FUNCTION_BLOCK REGRESS_OUT (* HMI elements for outputs of a REGRESS instance *)
  (* Standard: IEC 61499; Classification: HMI; Function: Output; Type: Linear Regression *)
  (* Version 0.0, 2006-07-20, JHC, Holobloc Inc *)
  (* Compiler header: package fb.rt.hmi; *)
  (* Compiler Java Sun JDK 1.5.0 *)
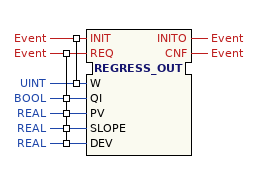
  EVENT_INPUT
    INIT WITH W; (* Initialization Request *)
    REQ WITH QI, PV, SLOPE, DEV; (* Request to Display Data *)
  END_EVENT
  EVENT_OUTPUT
    INITO; (* Initialization Confirm *)
    CNF; (* Data Display Confirmation *)
  END_EVENT
  VAR_INPUT
    W : UINT := 10; (* Text field width in characters *)
    QI : BOOL; (* Sample buffer full, outputs valid *)
    PV : REAL; (* Projected next value of regressed data *)
    SLOPE : REAL; (* Slope of regressed data, IN units per clock period. *)
    DEV : REAL; (* Estimated standard deviation from regression line *)
  END_VAR
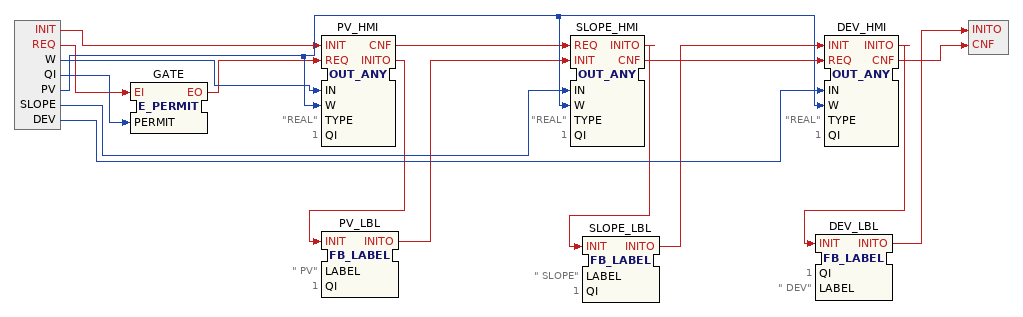
  FBS
    GATE : E_PERMIT; (* Only display valid data *)
    PV_HMI : OUT_ANY(TYPE := "REAL", QI := 1);
    SLOPE_HMI : OUT_ANY(TYPE := "REAL", QI := 1);
    DEV_HMI : OUT_ANY(TYPE := "REAL", QI := 1);
    PV_LBL : FB_LABEL(LABEL := " PV", QI := 1);
    SLOPE_LBL : FB_LABEL(LABEL := " SLOPE", QI := 1);
    DEV_LBL : FB_LABEL(QI := 1, LABEL := " DEV");
  END_FBS
  EVENT_CONNECTIONS
    REQ TO GATE.EI;
    INIT TO PV_HMI.INIT;
    DEV_LBL.INITO TO INITO;
    GATE.EO TO PV_HMI.REQ;
    PV_HMI.CNF TO SLOPE_HMI.REQ;
    PV_HMI.INITO TO PV_LBL.INIT;
    PV_LBL.INITO TO SLOPE_HMI.INIT;
    SLOPE_HMI.INITO TO SLOPE_LBL.INIT;
    SLOPE_LBL.INITO TO DEV_HMI.INIT;
    SLOPE_HMI.CNF TO DEV_HMI.REQ;
    DEV_HMI.INITO TO DEV_LBL.INIT;
    DEV_HMI.CNF TO CNF;
  END_CONNECTIONS
  DATA_CONNECTIONS
    QI TO GATE.PERMIT;
    PV TO PV_HMI.IN;
    SLOPE TO SLOPE_HMI.IN;
    DEV TO DEV_HMI.IN;
    W TO PV_HMI.W;
    W TO SLOPE_HMI.W;
    W TO DEV_HMI.W;
  END_CONNECTIONS
END_FUNCTION_BLOCK
